TYPE ARCommunicationSendPacketValueStore_t :
UNION
	valueString : STRING(255);
	valueInt : INT;
	valuebool : BOOL;
END_UNION
END_TYPE

(* stored: Version 1.1.0.1
   DUT ARCommunicationSendPacketValueStore_t: Id {855ca8e3-8182-4faa-a52f-f2825afa343f} *)
